FUNCTION_BLOCK F_LREAL_TO_UINT (* Convert LREAL to UINT *)
  (* Standard: 61499-1; Description: Copyright (c) 2023 Martin Erich Jobst This program and the accompanying materials are made available under the terms of the Eclipse Public License 2.0 which is available at https://www.eclipse.org/legal/epl-2.0/ SPDX-License-Identifier: EPL-2.0 *)
  (* Version 1.0, 2023-04-28, Martin Jobst *)
  (* Version 3.0, 2025-04-14, Patrick Aigner, changed package *)
  PACKAGE iec61131::conversion;
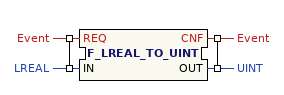
  EVENT_INPUT
    REQ WITH IN; (* Normal Execution Request *)
  END_EVENT
  EVENT_OUTPUT
    CNF WITH OUT; (* Execution Confirmation *)
  END_EVENT
  VAR_INPUT
    IN : LREAL;
  END_VAR
  VAR_OUTPUT
    OUT : UINT;
  END_VAR
  ALGORITHM REQ IN ST:
OUT := LREAL_TO_UINT(IN);
  END_ALGORITHM
END_FUNCTION_BLOCK
